{attribute 'qualified_only'}
{attribute 'strict'}
{attribute 'to_string'}
TYPE
    eMachineStatus :
    (

        Blue     := 100,
        White    := 200,
        Violet   := 300,
        Turquise := 400,
        All      := 990
    ) INT;
END_TYPE

(* stored: Version 1.1.0.1, ProductVersion 3.1.4024.12
   DUT eMachineStatus: Id {3313c827-6ec7-0a50-030a-1616b65e8e1d} *)
